# EPICS StreamDevice protocol: agilent33521aApp/db/agilent33521a.proto
TERMINATOR = NL;
ExtraInput = Ignore;
ReplyTimeout = 1000;

channelOutputRead {
    out "OUTPut1?";
    in "%i"
}

channelOutputEnable {
    out "OUTPut1 %{OFF|ON}";
    @init { channelOutputRead; }
}

getWaveformFunction {
    out "SOURce1:FUNCtion?";
    in "%{SIN|SQU|TRI|RAMP|PULS|PRBS|NOIS|ARB|DC}"
}

setWaveformFunction {
    out "SOURce1:FUNCtion %{SIN|SQU|TRI|RAMP|PULS|PRBS|NOIS|ARB|DC}";
    @init { getWaveformFunction }
}

getFrequency {
    out "SOURce1:FREQuency?";
    in "%f";
    @init { wait 5000; }
}

setFrequency {
    out "SOURce1:FREQuency %f";
    @init { getFrequency }
}

getAmplitude {
    out "SOURce1:VOLT?";
    in "%f";
}

setAmplitude {
    out "SOURce1:VOLT %f";
    @init { getAmplitude }
}

getOffset {
    out "SOURce1:VOLT:OFFSet?";
    in "%f"
}

setOffset {
    out "SOURce1:VOLT:OFFSet %f";
    @init { getOffset }
}

getPhase {
    out "SOURce1:PHASe?";
    in "%f"
}

setPhase {
    out "SOURce1:PHASe %f";
    @init { getPhase }
}

getSquareDutyCycle {
    out "SOURce1:FUNCtion:SQUare:DCYCle?";
    in "%f"
}

setSquareDutyCycle {
    out "SOURce1:FUNCtion:SQUare:DCYCle %f";
    @init { getSquareDutyCycle }
}

getRampSymmetry {
    out "SOURce1:FUNCtion:RAMP:SYMMetry?";
    in "%f"
}

setRampSymmetry {
    out "SOURce1:FUNCtion:RAMP:SYMMetry %f";
    @init { getRampSymmetry }
}

getPulseWidth {
    out "SOURce1:FUNCtion:PULSe:WIDTh?";
    in "%f"
}

setPulseWidth {
    out "SOURce1:FUNCtion:PULSe:WIDTh %f";
    @init { getPulseWidth }
}

getPulseLeadingEdge {
    out "SOURce1:FUNCtion:PULSe:TRANsition:LEADing?";
    in "%f"
}
